{attribute 'GeneratedUsingTerminal: EL6614-0000-0016'}
{attribute addProperty BoxType "EL6614-0000-0016"}
{attribute addProperty Id "InfoDataAT %I*InfoData_94A18F5E2"}
{attribute addProperty CRC "2009557638"}
{attribute addProperty Size "2"}
TYPE EL6614_77C76A86 EXTENDS EtcSlaveTerminalBase_947E5A46 :
STRUCT
	{attribute addProperty Name "InfoData"}
	InfoData : InfoData_94A18F5E;
END_STRUCT
END_TYPE

(* stored: Version 1.2.0.0, ProductVersion 3.1.4024.9
   DUT EL6614_77C76A86: Id {16b34028-b2a1-4c2d-bb8b-1a1818e58119} *)
